Staubli VAL3: StaubliSocket.pjx

--- StaubliSocket.pjx ---
Parameters version=s7.7 stackSize=5000 millimeterUnit=true
Program file=ReadMe.pgx
Program file=ServerGet.pgx
Program file=ServerSend.pgx
Program file=Task4ms.pgx
Program file=start.pgx
Program file=stop.pgx
Data file=StaubliSocket.dtx

--- StaubliSocket.dtx ---
bool bBool
jointRs jJRs
jointRx jJ
mdesc mNomSpeed
num nPcNum[6]
sio sServer = {link=Socket\clserver}
string sPos

--- start.pgx ---
program start()
  local num l_ncIoStatus
  local num l_nsIoStatus
  local string l_sMess
begin
  //-----------------------------------------------------------------------
  //Header begin
  //Description of program
  // 对套接字socket的客户端和服务器进行发送与接收信息
  //Input parameters
  //
  //Output paramaters
  //Example
  // 直接运行
  //History
  //  Creation : 2014.1.26 y.ye@staubli.com
  //Header end
  //-----------------------------------------------------------------------
  //运行程序注意事项：
  //先运行SOCKET程序上的服务器，然后在运行val3 staubliSocket,
  //再连接socket程序的客户端


  //界面初始化
  cls()
  title("测试Socket通讯:")
  gotoxy(1,1)
  put("程序已经运行:")
  userPage()

  //  //客户端
  //  l_ncIoStatus=ioStatus(sClient)
  //  gotoxy(1,3)
  //  put("客户端状态:"+toString("",l_ncIoStatus)+"      ")

  //服务器
  l_nsIoStatus=ioStatus(sServer)
  gotoxy(1,4)
  put("服务器状态:"+toString("",l_nsIoStatus)+"      ")

  //判断状态
  if l_ncIoStatus!=0
    popUpMsg("套接字不正确")
    return
  endIf

  //没有ClearBuffer 这个比较难联通
  clearBuffer(sServer)

  //同步任务建立
  taskCreateSync "TIME",0.004,bBool,Task4ms()



end

--- ClientSend.pgx ---
public program ClientSend(string x_sMess)
begin
  sClient=x_sMess
end

--- ReadMe.pgx ---
program ReadMe()
begin
  //对于Socket的客户端与服务器
  //可以使用Val3语言进行配置与可以

  //1.USR/configs/sio.cfx进行配置
  //2.在menu/控制面板/输入输出/接口列表中进行自定义配置


  //客户端要配置所要链接的服务器的IP和端口

  //服务器要配置端口

  //当sio.cfx进行配置好

  //同一个机器人上客户端的IP不要设为127.0.0.1 否则容易形成内环


  //sio.cfx格式
  //  <?xml version="1.0" encoding="utf-8" ?>
  //<sio>
  //  <socketClt>
  //    <String name="name" value="StlClient" />
  //    <String name="desc" value="" />
  //    <Inet name="serverIp" value="127.0.0.1" />
  //    <Uint name="portNumber" value="1000" />
  //    <Int name="endOfString" value="20" />
  //    <Float name="timeOut" value="0" />
  //    <Bool name="nagle" value="true" />
  //  </socketClt>
  //  <socketSrv>
  //    <String name="name" value="StlServer" />
  //    <String name="desc" value="" />
  //    <Uint name="portNumber" value="2000" />
  //    <Int name="endOfString" value="13" />
  //    <Float name="timeOut" value="5" />
  //    <Bool name="nagle" value="true" />
  //  </socketSrv>
  //</sio>

















end

--- ServerGet.pgx ---
public program ServerGet(string& x_sRes (dimensions=1))
  local num l_nIndex
  local num l_nNum[200]
begin
  x_sRes=""

  //从服务器获得字符串
  //  if sioGet(sServer,l_nNum)<0
  //    return
  //  endIf
  wait(sioGet(sServer,l_nNum)>=0)


  //把Acsii转换为字符串
  for l_nIndex=0 to size(l_nNum)-1
    x_sRes=x_sRes+chr(l_nNum[l_nIndex])
  endFor

end

--- stop.pgx ---
program stop()
begin
  cls()
  gotoxy(10,5)
  put("欢迎再次使用!")

end

--- Task4ms.pgx ---
program Task4ms()
  local bool l_bBool
  local num l_nNum
  local string l_sMess
  local string l_sS
begin


  resetMotion()
  cls()


  //把客户端收到不为空的信息通过服务器传送出去

  mNomSpeed.blend=off
 // $movejSyncBegin(mNomSpeed)
  while true
    //获取当前的关节值

    jJ=$getJntFbk()

    l_sMess=toString(".3",clock())+":"+toString(".3",jJ.j1)+","+toString(".3",jJ.j2)+","+toString(".3",jJ.j3)+","+toString(".3",jJ.j4)+","+toString(".3",jJ.j5)+","+toString(".3",jJ.j6)
    //发送数据
    call ServerSend(l_sMess)
    //收发位置
    call ServerGet(l_sMess)
    //在屏幕上显示
    if l_sMess!="" and find(l_sMess,",")>0

      //打印出来
      userPage()
      gotoxy(1,5)
      put("服务器端收到PC信息:")
      gotoxy(1,6)
      put(l_sMess+"             ")

      //2014.12.24
      //

      //***************************
      //分割数据
      l_nNum=0
      while find(l_sMess,",")>0
        l_sS=left(l_sMess,find(l_sMess,","))
        l_sMess=right(l_sMess,len(l_sMess)-len(l_sS)-1)
        toNum(l_sS,nPcNum[l_nNum],l_bBool)
        if !l_bBool
          disablePower()
        endIf
        l_nNum=l_nNum+1
      endWhile
      //***************************

      jJ.j1=nPcNum[0]
      jJ.j2=nPcNum[1]
      jJ.j3=nPcNum[2]
      jJ.j4=nPcNum[3]
      jJ.j5=nPcNum[4]
      jJ.j6=nPcNum[5]


     // $movejSync(jJ)







      //
    endIf
    delay(0)
  endWhile
 // $movejSyncEnd()




end
